// TIA Portal V16 export
// export: Created 2021-11-12T13:32:47.9647303Z, ExportSetting WithDefaults, DisplayName Totally Integrated Automation Portal, DisplayVersion V16 Update 3, DisplayName TIA Portal Version Control Interface, DisplayVersion V16 Update 2, DisplayName TIA Portal Openness, DisplayVersion V16 Update 3, DisplayName SINAMICS Startdrive Advanced, DisplayVersion V16 Update 5, DisplayName SINAMICS Startdrive G130, G150, S120, S150, SINAMICS MV, S210, DisplayVersion V16 Update 5, DisplayName SINAMICS Startdrive G110M, G120, G120C, G120D, G120P, G115D, DisplayVersion V16 Update 5, DisplayName STEP 7 Professional, DisplayVersion V16 Update 3, DisplayName STEP 7 Safety, DisplayVersion V16, DisplayName WinCC UA Professional, DisplayVersion V16 Update 3
DATA_BLOCK "STATUS_330"   // DB82
{ S7_Optimized_Access := 'TRUE' }
VERSION : 0.1
// stored: AutoNumber true, DBAccessibleFromOPCUA true, IsOnlyStoredInLoadMemory false, IsRetainMemResEnabled false, IsWriteProtectedInAS false, MemoryReserve 100
   VAR
      xxxxx___BinarySensors___xxxxx : Byte;
      "GL01-BG01" : Bool;   // Reflexní optická závora - Snímání pohybu dílu na dopravníku
      "GL01-BG02" : Bool;   // Reflexní optická závora - do CL01
      "GL02-BG01" : Bool;   // Reflexní optická závora - Snímání pohybu dílu na dopravníku
      "GL03-BG01" : Bool;   // Reflexní optická závora - Snímání pohybu dílu na dopravníku
      "UC21-FC01_14" : Bool;   // 400V Dopravník ++330 (MK1) OK
      "UC21-FC02_14" : Bool;   // 400V Dopravník ++330 (MK2) OK
      "UC21-FC03_14" : Bool;   // 400V Dopravník ++330 ( MK3) OK
      xxxxx___BinaryOthers___xxxxx : Byte;
      "UH11-SF01_14" : Bool;   // Conveyor Remote
      "UH11-SF01_24" : Bool;   // Conveyor Automat
      "UH11-SF03_14" : Bool;   // Conveyor Start automat
      "UH11-SF04_12" : Bool;   // Conveyor Stop
      "UH11-SF05_14" : Bool;   // Conveyor GL01 Manual Backward
      "UH11-SF05_24" : Bool;   // Conveyor GL01 Manual Forward
      "UH11-SF06_14" : Bool;   // Conveyor GL02 Manual Backward
      "UH11-SF06_24" : Bool;   // Conveyor GL02 Manual Forward
      "UF01-SF02_14" : Bool;   // Conveyor GL03 Manual Backward
      "UF01-SF02_24" : Bool;   // Conveyor GL03 Manual Forward
      "UH11-SF07_14" : Bool;   // Bedna Žádost o výměnu
      "UH11-SF08_14" : Bool;   // Bedna vyměněna
      xxxxx___Drives___xxxxx : Byte;
      "GL01-MA01" : Struct   // Conveyour to oldering furnace (MK1) - drive / Dopravník do stárnoucí pece (MK1) - motor
         Main { S7_SetPoint := 'True'} : "UDT_Status_main";
         Specific { S7_SetPoint := 'True'} : "UDT_Drive1_Status_specific";
         Error { S7_SetPoint := 'True'} : "UDT_Error01";
      END_STRUCT;
      "GL02-MA01" : Struct   // Conveyour to oldering furnace (MK2) - drive / Dopravník do stárnoucí pece (MK2) - motor
         Main { S7_SetPoint := 'True'} : "UDT_Status_main";
         Specific { S7_SetPoint := 'True'} : "UDT_Drive1_Status_specific";
         Error { S7_SetPoint := 'True'} : "UDT_Error01";
      END_STRUCT;
      "GL03-MA01" : Struct   // Conveyour to oldering furnace (MK3) - drive / Dopravník do stárnoucí pece (MK3) - motor
         Main { S7_SetPoint := 'True'} : "UDT_Status_main";
         Specific { S7_SetPoint := 'True'} : "UDT_Drive1_Status_specific";
         Error { S7_SetPoint := 'True'} : "UDT_Error01";
      END_STRUCT;
      "UC21-TA01" : Struct   // Conveyour to oldering furnace (MK1) - G120 / Dopravník do stárnoucí pece (MK1) - měnič G120
         Main { S7_SetPoint := 'True'} : "UDT_Status_main";
         Specific { S7_SetPoint := 'True'} : "UDT_SINAMICS_G120_Status_specific";
         Error { S7_SetPoint := 'True'} : "UDT_Error02";
      END_STRUCT;
      "UC21-TA02" : Struct   // Conveyour to oldering furnace (MK2) - G120 / Dopravník do stárnoucí pece (MK2) - měnič G120
         Main { S7_SetPoint := 'True'} : "UDT_Status_main";
         Specific { S7_SetPoint := 'True'} : "UDT_SINAMICS_G120_Status_specific";
         Error { S7_SetPoint := 'True'} : "UDT_Error02";
      END_STRUCT;
      "UC21-TA03" : Struct   // Conveyour to oldering furnace (MK3) - G120 / Dopravník do stárnoucí pece (MK3) - měnič G120
         Main { S7_SetPoint := 'True'} : "UDT_Status_main";
         Specific { S7_SetPoint := 'True'} : "UDT_SINAMICS_G120_Status_specific";
         Error { S7_SetPoint := 'True'} : "UDT_Error02";
      END_STRUCT;
      xxxxx__Others__xxxxx : Byte;
      CL01 : Struct   // Box for NOK parts / Bedna na NOK kusy
         Main : "UDT_Status_main";
         Specific : "UDT_PartCounter_Status";
         Error : "UDT_Error01";
      END_STRUCT;
      xxxxx__Alarms__xxxxx : Byte;
      CL01_Warn : Struct   // Box full warning / Bedna plná.
         Main : "UDT_Status_main";
         Specific { S7_SetPoint := 'True'} : "UDT_DI_Mon_Status_specific";
         Error { S7_SetPoint := 'True'} : "UDT_Error01";
      END_STRUCT;
      CL01_Alarm : Struct   // Box full alarm / Bedna plná.
         Main : "UDT_Status_main";
         Specific : "UDT_DI_Mon_Status_specific";
         Error : "UDT_Error01";
      END_STRUCT;
      ES : Struct   // E-stop
         Main { S7_SetPoint := 'True'} : "UDT_Status_main";
         Specific { S7_SetPoint := 'True'} : "UDT_DI_Mon_Status_specific";
         Error { S7_SetPoint := 'True'} : "UDT_Error01";
      END_STRUCT;
   END_VAR
BEGIN
END_DATA_BLOCK
